PROGRAM FB_CPUDiagnosatics
VAR
	bExecute 				: BOOL;
	tPeriod 				: TIME := T#500MS ;
	fbReadIPCDiagnostics 	: FB_IPCDiag_ReadParameterPeriodic 	;
	eParameterKey			: E_IPCDiag_ParameterKey			;
END_VAR
VAR_IN_OUT
	fbDiagRegister			: FB_IPCDiag_Register ;
END_VAR

END_PROGRAM

(* stored: Version 1.1.0.1
   POU FB_CPUDiagnosatics: Id {5b14e865-572c-476c-b156-e10f10f57ed2}, SpecialFunc None *)
